PROGRAM prgComEffIO
VAR
	fbCom		: FB_MqttCommunicator_V3;
END_VAR

fbCom(
	bConnect				:= TRUE,
	strAuthKey				:=  'BMS99299754422' , 
	sUserName				:= '3e50e6d5-eb07-43c8-8301-26b96effcdd6', 
	sUserPassword			:= '00b28941-9e96-4cb2-9f19-540a3e4b2bd2', 
	eSavePositionCertificate:= eSavePositionOnPLC.ePostionHardDisk, 
	time_HeartBeat_sec := T#15S,
	bConnected=> , 
	bError=> , 
	hrErrorCode=> , 
	eConnectionState=> , 
	eErrorMessage_Out=> );

END_PROGRAM

(* stored: Version 1.1.0.1, ProductVersion 3.1.4024.12
   POU prgComEffIO: Id {cbcd318b-bf51-484c-bcaa-d6efcdf43fe3}, SpecialFunc None *)
